{attribute 'pack_mode':='1'}
TYPE SwapToteParams :
STRUCT
   source_id : ModelIdentifier;
   working_id : ModelIdentifier; 
   outbound_id : ModelIdentifier; 
END_STRUCT
END_TYPE

(* stored: Version 1.1.0.1, ProductVersion 3.1.4024.12
   DUT SwapToteParams: Id {68363950-9687-4428-85f5-853cb8ad7dcf} *)
